// TIA Portal V19 export
DATA_BLOCK "A02_MwFacCalc_Gripper"   // DB4, Motion_DB
// stored: InstanceOfName TO_ExternalEncoder, OfSystemLibElement TO_ExternalEncoder, OfSystemLibVersion 8.0
TO_ExternalEncoder   // technology object, version 8.0
// stored: Connection Interface Sensor, SensorIndexInActorTelegram 1, PathToDBMember Encoder.1248A1.Sensor_1
   // // inherited from TO_Axis
   // // inherited from TO_Object
   // VAR
   //    ActualPosition { ExternalWritable := 'False'} : LReal;
   //    ActualVelocity { ExternalWritable := 'False'} : LReal;
   //    ActualAcceleration { ExternalWritable := 'False'} : LReal;
   //    ActualModuloCycle { ExternalWritable := 'False'} : DInt;
   //    Sensor { S7_SetPoint := 'True'} : TO_Struct_ExternalEncoder_Sensor;
   //    CrossPlcSynchronousOperation { S7_SetPoint := 'True'} : TO_Struct_CrossPlcSynchronousOperation;
   //    Extrapolation { S7_SetPoint := 'True'} : TO_Struct_Extrapolation;
   //    Mechanics { S7_SetPoint := 'True'} : TO_Struct_Mechanics;
   //    LoadGear { S7_SetPoint := 'True'} : TO_Struct_LoadGear;
   //    Properties { ExternalWritable := 'False'; S7_SetPoint := 'True'} : TO_Struct_Properties;
   //    Modulo { S7_SetPoint := 'True'} : TO_Struct_Modulo;
   //    Homing { S7_SetPoint := 'True'} : TO_Struct_ExternalEncoder_Homing;
   //    StandstillSignal { S7_SetPoint := 'True'} : TO_Struct_StandstillSignal;
   //    Units { ExternalWritable := 'False'; S7_SetPoint := 'True'} : TO_Struct_ExternalEncoder_Units;
   //    StatusProvidedLeadingValue { ExternalWritable := 'False'; S7_SetPoint := 'True'} : TO_Struct_StatusProvidedLeadingValue;
   //    StatusSensor { ExternalWritable := 'False'; S7_SetPoint := 'True'} : TO_Struct_StatusSensor;
   //    StatusExtrapolation { ExternalWritable := 'False'; S7_SetPoint := 'True'} : TO_Struct_StatusExtrapolation;
   //    StatusWord { ExternalWritable := 'False'} : DWord;
   //    ErrorWord { ExternalWritable := 'False'} : DWord;
   //    ErrorDetail { ExternalWritable := 'False'; S7_SetPoint := 'True'} : TO_Struct_ErrorDetail;
   //    WarningWord { ExternalWritable := 'False'} : DWord;
   //    InternalToTrace { S7_SetPoint := 'True'} : Array[1..4] of TO_Struct_Internal;
   // END_VAR
BEGIN
   Sensor.InverseDirection := true;
   Sensor.System := 0;
   Sensor.Interface.AddressIn.RID := 16#208070e;
   Sensor.Interface.AddressIn.AREA := 16#8b;
   Sensor.Interface.AddressIn.DB_NUMBER := 160;
   Sensor.Interface.AddressIn.OFFSET := 32;
   Sensor.Interface.AddressOut.RID := 16#208070f;
   Sensor.Interface.AddressOut.AREA := 16#8b;
   Sensor.Interface.AddressOut.DB_NUMBER := 160;
   Sensor.Interface.AddressOut.OFFSET := 352;
   Sensor.Parameter.Resolution := 0.004;
   _Sensor.Interface.Telegram := 81;
END_DATA_BLOCK
